// TIA Portal V20 export
DATA_BLOCK "DB_HMICmd"   // DB86
{ S7_Optimized_Access := 'TRUE' }
// stored: MemoryReserve 100
   VAR
      IntGateCloseReq : Bool;
      IntGateOpenReq : Bool;
      ExtGateCloseReq : Bool;
      ExtGateOpenReq : Bool;
      IntGateCloseCmd : Bool;
      IntGateOpenCmd : Bool;
      ExtGateCloseCmd : Bool;
      ExtGateOpenCmd : Bool;
      BlowingCmd : Bool;
   END_VAR
BEGIN
END_DATA_BLOCK
